// Mitsubishi GX Works2 project: 240430_timechart05_병렬회로gxw   PLC: Q03UDV

PROGRAM MAIN
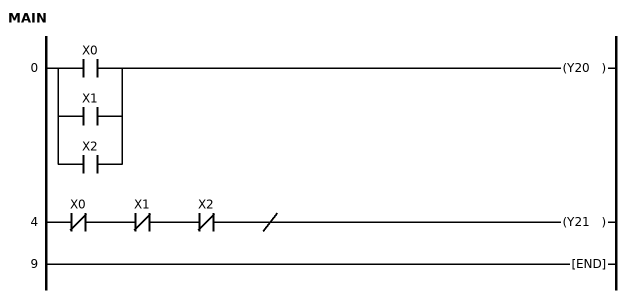
0     LD      X0
      OR      X1
      OR      X2
      OUT     Y20
4     LDI     X0
      ANI     X1
      ANI     X2
      INV
      OUT     Y21
9     END
END_PROGRAM
